{attribute 'OPC.UA.DA' := '1'}
FUNCTION_BLOCK FB_Valve_ONOFF_woMonitoring_1 EXTENDS FB_BaseDevice IMPLEMENTS I_Device, I_ValveActuated

VAR
	
	{attribute 'OPC.UA.DA' := '1'} 
	bValveMonitor_OPEN AT %I*: BOOL := FALSE;
	{attribute 'OPC.UA.DA' := '1'} 
	bValveMonitor_CLOSED AT %I*: BOOL := FALSE;
	{attribute 'OPC.UA.DA' := '1'} 
	bValveOutput_OPEN AT %Q*: BOOL := FALSE;
	{attribute 'OPC.UA.DA' := '1'} 
	bValveOutput_CLOSE AT %Q*: BOOL := FALSE;
	
	{attribute 'OPC.UA.DA' := '0'} 
	eSMState: (WAIT, CLOSING, CLOSED, OPENING, OPEN);
	
	{attribute 'OPC.UA.DA' := '1'} 
	tActionTimeout: TIME := T#5S;
	{attribute 'OPC.UA.DA' := '0'} 
	fbTON_timeout: TON := (PT := tActionTimeout, IN := FALSE);
	{attribute 'OPC.UA.DA' := '0'}
	fbTON_simulation_delay: TON := (PT := T#1S, IN := FALSE);
END_VAR

fbTONstartTime();
fbTONstopTime();

IF GVL.bAutoUpdateDeviceState THEN
	eState := eStateTarget;	
END_IF

IF bEnable = FALSE THEN
	eSMState := CLOSE
END_IF

	
CASE eSMState OF
	
	WAIT:
		//Wait for method call to change ESMState
		
	OPENING: 
		eState := E_DeviceState.TURNING_ON;
		bValveOutput_CLOSE 	:= FALSE;
		bValveOutput_OPEN 	:= TRUE;

	
		IF fbTONstartTime.Q THEN
			eSMState := WAIT;
			raiseAlarm(Priority := E_AlarmPriority.High, Label := 'Failed to Open', Enabled := TRUE, DeviceAlarmID := 1);
		END_IF
		
		IF bValveMonitor_OPEN  THEN
			eSMState := OPEN;
			eState := E_DeviceState.OPEN;
		END_IF
		
	OPEN:
		IF bValveMonitor_OPEN <> TRUE THEN
			raiseAlarm(Priority := E_AlarmPriority.High, Label := 'Valve Closed Unexpectedly', Enabled := TRUE, DeviceAlarmID := 2);
			eState := E_DeviceState.CLOSED;
			eSMState := WAIT;
		END_IF
		

	CLOSING:
		eState := E_DeviceState.TURNING_OFF;
		bValveOutput_CLOSE 	:= TRUE;
		bValveOutput_OPEN 	:= FALSE;

				
		IF fbTONstopTime.Q THEN
			eSMState := WAIT;
			raiseAlarm(Priority := E_AlarmPriority.High, Label := 'Failed to Close', Enabled := TRUE, DeviceAlarmID := 3);
		END_IF 
		
		IF bValveMonitor_CLOSED = TRUE THEN
			eSMState := CLOSED;	
		END_IF
		

	CLOSED:
		eState := E_DeviceState.CLOSED;
		eSMState := WAIT;
		
END_CASE

{warning 'add method implementation '}
METHOD close : BOOL
eSMState := CLOSING;
END_METHOD

{warning 'add method implementation '}
METHOD disable : BOOL
bEnable := FALSE;
END_METHOD

{warning 'add method implementation '}
METHOD enable : BOOL
bEnable := TRUE;
END_METHOD

{warning 'add method implementation '}
METHOD FB_init : BOOL
VAR_INPUT
	(* if TRUE, the retain variables are initialized (warm start / cold start)*)
	bInitRetains	: BOOL;
	(* if TRUE, the instance afterwards gets moved into the copy code (online change)*)
	bInCopyCode	: BOOL;
	
	ValveID: STRING(80);
	ValveDescr: STRING(255); 
END_VAR
sID := ValveID;
sDescr := ValveDescr;
END_METHOD

{warning 'add method implementation '}
METHOD open : BOOL
eSMState := OPENING;
END_METHOD

END_FUNCTION_BLOCK

(* stored: Version 1.1.0.1, ProductVersion 3.1.4024.12
   POU FB_Valve_ONOFF_woMonitoring_1: Id {381ecdce-874b-45df-befe-2affcb9f55dc}, SpecialFunc None
   Method close: Id {7bf9648b-f4d0-471b-9726-f9d18b0fcb72}
   Method disable: Id {20b18462-0c10-4d61-b2f1-7a189a821346}
   Method enable: Id {977408f2-4580-46e6-a693-706688e61fc0}
   Method FB_init: Id {2a3fb5bb-98a9-4870-b7b0-7534d171ef8b}
   Method open: Id {08a2afaf-59a1-4b47-a8c8-bb1e63b6e563} *)
